# EPICS autosave request: ADApp/Db/NDCentroid_settings.req
$(P)$(R)ComputeCentroid
$(P)$(R)CentroidThreshold
